// TIA Portal V17 export
// export: Created 2026-04-13T11:12:41.9894962Z, ExportSetting WithDefaults, DisplayName Totally Integrated Automation Portal, DisplayVersion V17 Update 4, DisplayName TIA Portal Openness, DisplayVersion V17 Update 4, DisplayName TIA Portal Version Control Interface, DisplayVersion V17, DisplayName SINAMICS Startdrive Advanced, DisplayVersion V17, DisplayName SINAMICS Startdrive G130, G150, S120, S150, SINAMICS MV, S210, DisplayVersion V17, DisplayName SINAMICS Startdrive G110M, G120, G120C, G120D, G120P, G115D, DisplayVersion V17, DisplayName STEP 7 Professional, DisplayVersion V17 Update 4, DisplayName STEP 7 Safety, DisplayVersion V17, DisplayName WinCC Professional, DisplayVersion V17 Update 4
FUNCTION_BLOCK "单元模式"   // FB81, SCL
{ S7_Optimized_Access := 'TRUE' }
VERSION : 0.1
// stored: AutoNumber true, IsIECCheckEnabled false, IsRetainMemResEnabled false, MemoryReserve 100, SetENOAutomatically false, UDAEnableTagReadback false
   VAR
      第一动作中 : Bool;
      第二动作中 : Bool;
      动作信号 : Bool;
      estop : Bool;
      动作按钮 : Bool;
      动作超时 : Bool;
      动作条件 : Bool;
      动作到位 : Bool;
      动作输出 : Bool;
      手动模式 : Bool;
      自动模式 : Bool;
      超时 : TON_TIME;
      故障复位 : Bool;
      反馈信号 : Bool;
   END_VAR
BEGIN
   #动作信号 := #第一动作中 OR #第二动作中;
   #动作条件 := NOT #estop AND NOT #动作超时;
   IF ((#自动模式 AND #动作信号) OR (#手动模式 AND #动作按钮) OR #动作输出)
       AND #动作条件
       AND NOT #动作到位 THEN
       #动作输出 := 1;
   ELSE
       #动作输出 := 0;
   END_IF;

   #动作到位 := #反馈信号;

   #超时(IN:=(#动作输出 AND NOT #动作到位),
       PT:=T#5S);

   #动作超时 := #超时.Q OR (#动作超时 AND NOT #故障复位);
END_FUNCTION_BLOCK
